ABB RobotStudio station: Práctica5_inicio.rsstn

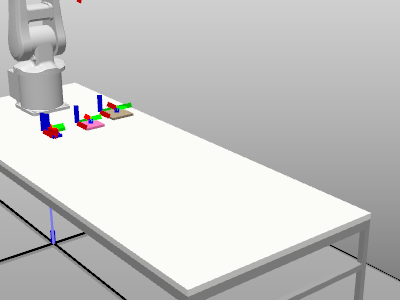
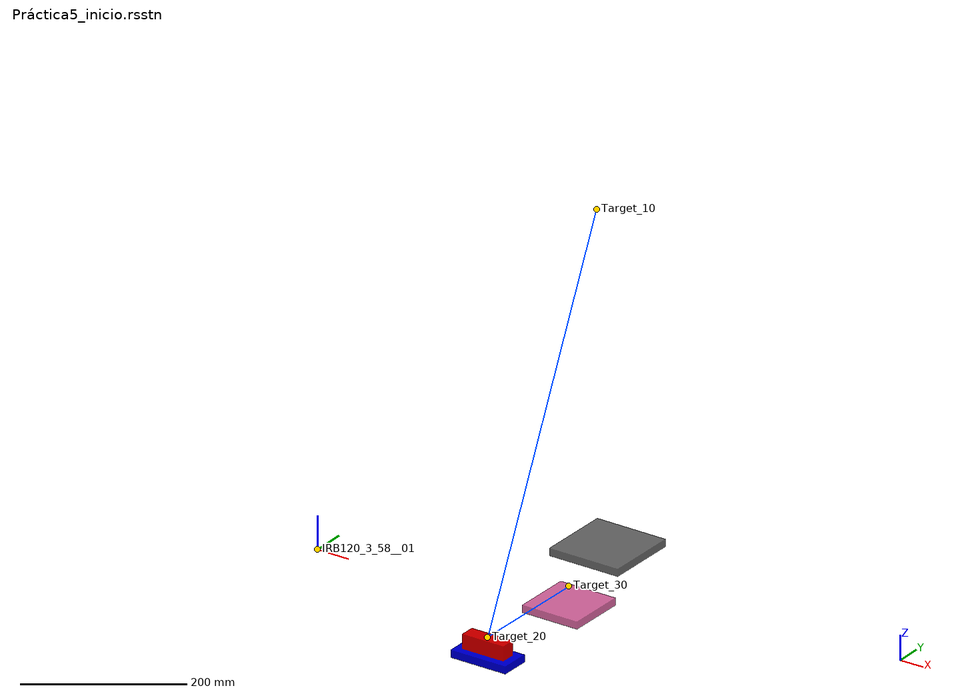
[picture v1: parts stored in the station drawn from their meshes, with robot base, taught points and paths (robot models come from the ABB library and are not in the file)]
Station Práctica3_inicio (saved by RobotStudio 25.1.11133.0)
Controller Controlador2, task T_ROB1: task frame (RAPID world) sits at (0, 0, 670) mm in the station
Controller Controlador2
  mechanical unit ROB_1: IRB120_3_58__01, 6 joints, base frame (0, 0, 0) mm
Layout (positions relative to the parent item):
  - TVentosa [mechanism] at (364.35, 0, 1264) mm, rotated rx 180 ry 60 rz 180 deg
      TCP TVentosa at (0, 0, 51.19) mm
      links: Mi_herramienta
  - LogicGate [smart component, from Components\LogicGate.rslib]
      properties: Operator=NOT; Delay=0
  - LogicGate_2 [smart component, from Components\LogicGate.rslib]
      properties: Operator=AND; Delay=0
  - IRB120_3_58__01 [mechanism, from %ABB.RobotStudio.Models.IRB120%\IRB120_3_58_G_01.rslib] at (0, 0, 670) mm; joint values [0, 0, 0, 0, 0.5236, 0] (rad or m)
  - table [part, from Libraries\e293a11e-ed86-4237-866f-a9bf8f4bd145table.rslib] at (-246.62, 300, 670) mm, rotated rx 0 ry 0 rz -90 deg
  - Base2 [part], size 80 x 80 x 10 mm
  - Base1 [part], size 80 x 40 x 10 mm
  - Detacher [smart component, from Components\Detacher.rslib]
      properties: Child=Pieza_1; KeepPosition=true
  - CollisionSensor [smart component, from Components\CollisionSensor.rslib]
      properties: Object1=TVentosa; Object2=Pieza_1; NearMiss=0.001; Part1=(none); Part2=(none); CollisionType=0
    - _sensorPart_ [part]
  - Attacher_2 [smart component, from Components\Attacher.rslib]
      properties: Parent=TVentosa; Flange=0; Child=Pieza_1; Mount=false; Offset=[0 0 0]; Orientation=[0 0 0]
  - Source_2 [smart component, from Components\Source.rslib]
      properties: Source=Pieza; Copy=Pieza_1; Parent=(none); Position=[0.34 -0.13 0.68]; Orientation=[0 0 0]; Transient=false; PhysicsBehavior=0
  - SimulationEvents_2 [smart component, from Components\SimulationEvents.rslib]
  - Pieza [part] at (340, -130, 700) mm, rotated rx 180 ry 0 rz 180 deg, size 60 x 20 x 20 mm
  - Pieza_2 [part], size 100 x 100 x 10 mm
  - Pieza_47 [part] at (340, -130, 680) mm, size 60 x 20 x 20 mm
  - Pieza_48 [part] at (340, -130, 680) mm, size 60 x 20 x 20 mm
  - Pieza_49 [part] at (340, -130, 680) mm, size 60 x 20 x 20 mm
  - Pieza_50 [part] at (340, -130, 680) mm, size 60 x 20 x 20 mm
  - Pieza_52 [part] at (340, -130, 680) mm, size 60 x 20 x 20 mm
  - Pieza_1 [part] at (340, -130, 680) mm, size 60 x 20 x 20 mm
Attachment: TVentosa is attached to IRB120_3_58__01 / Link6
Attachment: Base2 is attached to Base1
Attachment: Base1 is attached to table
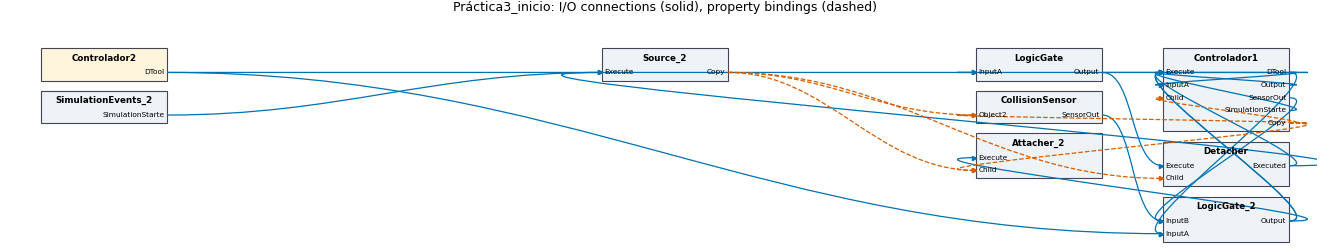
Station logic (signal -> signal, property => property):
  Controlador1.DTool -> Attacher.Execute
  Controlador1.DTool -> LogicGate_2.InputA
  LogicGate_2.Output -> Detacher.Execute
  Controlador1.DTool -> LogicGate.InputA
  LogicGate.Output -> Detacher.Execute
  CollisionSensor.SensorOut -> LogicGate_2.InputB
  Controlador1.DTool -> LogicGate_2.InputA
  LogicGate_2.Output -> Attacher.Execute
  Controlador2.DTool -> LogicGate.InputA
  LogicGate.Output -> Detacher.Execute
  Controlador2.DTool -> LogicGate_2.InputA
  LogicGate_2.Output -> Attacher.Execute
  Detacher.Executed -> Source.Execute
  SimulationEvents.SimulationStarted -> Source.Execute
  CollisionSensor.SensorOut -> LogicGate_2.InputB
  SimulationEvents_2.SimulationStarted -> Source_2.Execute
  Detacher.Executed -> Source_2.Execute
  LogicGate_2.Output -> Attacher_2.Execute
  Source.Copy => Attacher.Child
  Source.Copy => CollisionSensor.Object2
  Source.Copy => Attacher_2.Child
  Source_2.Copy => Attacher_2.Child
  Source_2.Copy => CollisionSensor.Object2
  Source_2.Copy => Detacher.Child
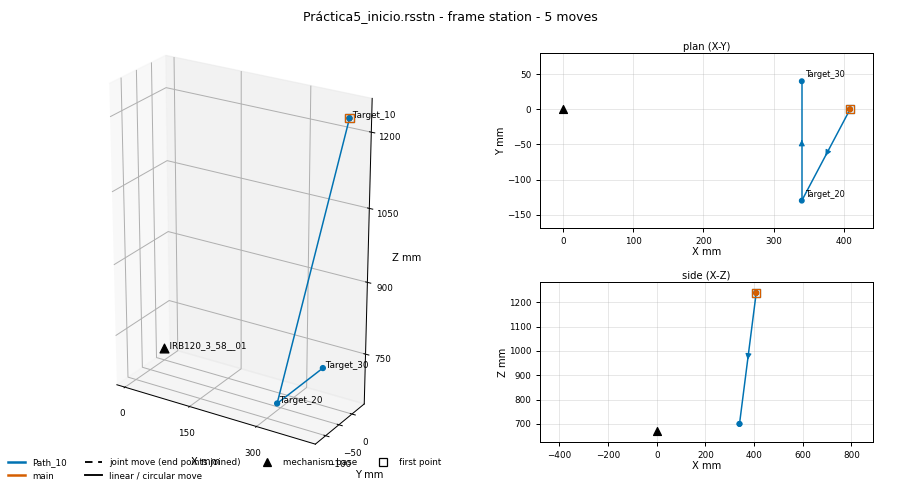
[picture p0: tool path of Práctica5_inicio.rsstn in frame station, 5 of 6 moves have a stored position in this frame; points joined in program order, loops and branches not executed]
Targets, tools, work objects and paths stored in the station, written as RAPID:
! task T_ROB1
MODULE CalibData
  PERS tooldata TVentosa:=[TRUE,[[0,0,51.19],[1,0,0,0]],[0.1,[0,0,1],[1,0,0,0],0,0,0]];
  TASK PERS wobjdata WO_Pieza:=[FALSE,TRUE,"",[[300,-150,10],[1,0,0,0]],[[20,10,0],[1,0,0,0]]];
  TASK PERS wobjdata WO_Base2:=[FALSE,TRUE,"",[[300,-150,10],[1,0,0,0]],[[0,150,0],[1,0,0,0]]];
  TASK PERS wobjdata CajonDesastre:=[FALSE,TRUE,"",[[237.224,146.16,10],[1,0,0,0]],[[50,50,20],[0,0,1,0]]];
  PROC Path_10()
    MoveJ Target_10,v200,z100,TVentosa\WObj:=wobj0;
    MoveL Target_20,v200,fine,TVentosa\WObj:=WO_Pieza;
    MoveL Target_30,v200,z100,TVentosa\WObj:=WO_Base2;
    MoveAbsJ JHome,v1000,z100,TVentosa\WObj:=WO_Pieza;
  ENDPROC
  PROC main()
    Initialize;
    MoveJ Target_10,v200,z100,TVentosa\WObj:=wobj0;
    MoveJ Target_10,v200,z100,TVentosa\WObj:=wobj0;
  ENDPROC
  PROC Initialize()
  ENDPROC
ENDMODULE

! task T_ROB1
MODULE Module1
  CONST robtarget Target_10:=[[408.685,0,568.405],[0.5,0,0.866025404,0],[0,0,0,0],[9E+09,9E+09,9E+09,9E+09,9E+09,9E+09]];
  CONST robtarget Target_20:=[[19.999989664,10.000006428,19.999948885],[-0.000000013,0,1,0.000000005],[-1,0,-1,0],[9E+09,9E+09,9E+09,9E+09,9E+09,9E+09]];
  CONST robtarget Target_30:=[[40,40,20],[0,0,1,0],[0,0,0,0],[9E+09,9E+09,9E+09,9E+09,9E+09,9E+09]];
  CONST jointtarget JHome:=[[0,0,-90,0,0,0],[9E+09,9E+09,9E+09,9E+09,9E+09,9E+09]];
  CONST robtarget Target_40:=[[0,0,0],[1,0,0,0],[0,0,0,0],[9E+09,9E+09,9E+09,9E+09,9E+09,9E+09]];
ENDMODULE

